GLOBALCONSTANTS bitconst (* Global constants *)
  (* Standard: 61499-1 *)
  (* Version 1.0, 2024-02-22, franz *)
  VAR_GLOBAL CONSTANT
    BOOL_BIT_ZZ : BOOL := 2#0; (* ZERO Constant *)
    BOOL_BIT_00 : BOOL := 2#1; (* Bit 00 Constant *)
    BYTE_BIT_ZZ : BYTE := 2#0000_0000; (* ZERO Constant *)
    BYTE_BIT_00 : BYTE := 2#0000_0001; (* Bit 00 Constant *)
    BYTE_BIT_01 : BYTE := 2#0000_0010; (* Bit 01 Constant *)
    BYTE_BIT_02 : BYTE := 2#0000_0100; (* Bit 02 Constant *)
    BYTE_BIT_03 : BYTE := 2#0000_1000; (* Bit 03 Constant *)
    BYTE_BIT_04 : BYTE := 2#0001_0000; (* Bit 04 Constant *)
    BYTE_BIT_05 : BYTE := 2#0010_0000; (* Bit 05 Constant *)
    BYTE_BIT_06 : BYTE := 2#0100_0000; (* Bit 06 Constant *)
    BYTE_BIT_07 : BYTE := 2#1000_0000; (* Bit 07 Constant *)
  END_VAR
END_GLOBALCONSTANTS
